FUNCTION_BLOCK MSDOC (* CAT Function Block Type *)
  (* Standard: 61499-2 *)
  (* Version 0.0, 6/7/2026, Schneider Electric, template *)
  PACKAGE SE.Nereda;
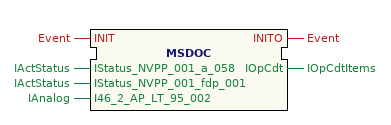
  EVENT_INPUT
    INIT;
  END_EVENT
  EVENT_OUTPUT
    INITO;
  END_EVENT
  SOCKETS
    IStatus_NVPP_001_a_058 : IActStatus;
    IStatus_NVPP_001_fdp_001 : IActStatus;
    I46_2_AP_LT_95_002 : IAnalog;
  END_SOCKETS
  PLUGS
    IOpCdt : IOpCdtItems;
  END_PLUGS
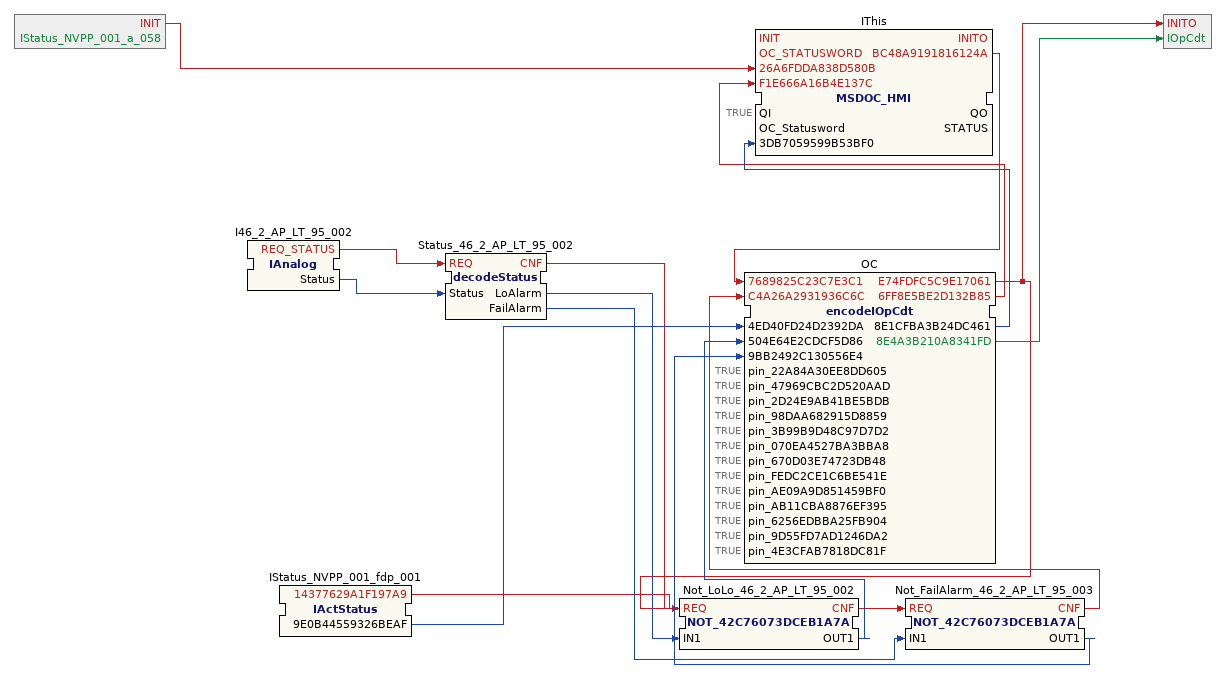
  (* 01 - FUNCTIONNAL INPUT INTERFACE *)
  (* 00 - INITIALIZATION *)
  (* 05 - LOGIC *)
  (* 06 - HMI INTERFACE *)
  (* 03 - FIELD INTERFACE *)
  (* Created by : Nouriddin OUECHEN 2026 *)
  (* Operating Condition Status *)
  (* Created by : Nouriddin OUECHEN 2026 *)
  (* 02 - FUNCTIONNAL OUTPUT INTERFACE *)
  (* Operating conditions : 2. No error from the metal salt dosing unit 3. No LL-level in the metal salt IBC 46 2 AP LT 95 002 4. Level measurement 46 2 AP LT 95 002 available *)
  FBS
    OC : encodeIOpCdt(pin_22A84A30EE8DD605 := TRUE, pin_47969CBC2D520AAD := TRUE, pin_2D24E9AB41BE5BDB := TRUE, pin_98DAA682915D8859 := TRUE, pin_3B99B9D48C97D7D2 := TRUE, pin_070EA4527BA3BBA8 := TRUE, pin_670D03E74723DB48 := TRUE, pin_FEDC2CE1C6BE541E := TRUE, pin_AE09A9D851459BF0 := TRUE, pin_AB11CBA8876EF395 := TRUE, pin_6256EDBBA25FB904 := TRUE, pin_9D55FD7AD1246DA2 := TRUE, pin_4E3CFAB7818DC81F := TRUE); (* You set the operating conditions. For the inputs that are not used set a constant to TRUE. *)
    IThis : MSDOC_HMI(QI := TRUE);
    Status_46_2_AP_LT_95_002 : decodeStatus; {SET_ATTRIBUTE(Configuration.Component.HideUnusedPorts, )}
    Not_LoLo_46_2_AP_LT_95_002 : NOT_42C76073DCEB1A7A; {SET_ATTRIBUTE(Configuration.GenericFBType.InterfaceParams, Runtime.Standard#CNT:=1;OUT${CNT$}:BOOL)}
    Not_FailAlarm_46_2_AP_LT_95_003 : NOT_42C76073DCEB1A7A; {SET_ATTRIBUTE(Configuration.GenericFBType.InterfaceParams, Runtime.Standard#CNT:=1;OUT${CNT$}:BOOL)}
  END_FBS
  EVENT_CONNECTIONS
    INIT TO IThis.26A6FDDA838D580B;
    OC.E74FDFC5C9E17061 TO INITO;
    OC.6FF8E5BE2D132B85 TO IThis.F1E666A16B4E137C;
    IThis.BC48A9191816124A TO OC.7689825C23C7E3C1;
    OC.E74FDFC5C9E17061 TO Not_LoLo_46_2_AP_LT_95_002.REQ;
    IStatus_NVPP_001_fdp_001.14377629A1F197A9 TO Not_LoLo_46_2_AP_LT_95_002.REQ;
    I46_2_AP_LT_95_002.REQ_STATUS TO Status_46_2_AP_LT_95_002.REQ;
    Not_FailAlarm_46_2_AP_LT_95_003.CNF TO OC.C4A26A2931936C6C;
    Not_LoLo_46_2_AP_LT_95_002.CNF TO Not_FailAlarm_46_2_AP_LT_95_003.REQ;
    Status_46_2_AP_LT_95_002.CNF TO Not_LoLo_46_2_AP_LT_95_002.REQ;
  END_CONNECTIONS
  DATA_CONNECTIONS
    OC.8E1CFBA3B24DC461 TO IThis.3DB7059599B53BF0;
    IStatus_NVPP_001_fdp_001.9E0B44559326BEAF TO OC.4ED40FD24D2392DA;
    I46_2_AP_LT_95_002.Status TO Status_46_2_AP_LT_95_002.Status;
    Status_46_2_AP_LT_95_002.LoAlarm TO Not_LoLo_46_2_AP_LT_95_002.IN1;
    Not_LoLo_46_2_AP_LT_95_002.OUT1 TO OC.504E64E2CDCF5D86;
    Status_46_2_AP_LT_95_002.FailAlarm TO Not_FailAlarm_46_2_AP_LT_95_003.IN1;
    Not_FailAlarm_46_2_AP_LT_95_003.OUT1 TO OC.9BB2492C130556E4;
  END_CONNECTIONS
  ADAPTER_CONNECTIONS
    OC.8E4A3B210A8341FD TO IOpCdt;
  END_CONNECTIONS
END_FUNCTION_BLOCK
